// Copyright (c) 2024 Loupe (https://loupe.team), provided under the MIT License.

INTERFACE IPLCopenCommand

METHOD Aborted : BOOL
VAR_INPUT
END_VAR
END_METHOD

METHOD AbortPreviousCommands : BOOL
VAR_INPUT
    newCommand : IPLCopenCommand;
END_VAR
END_METHOD

PROPERTY Consume : BOOL
GET
END_GET
END_PROPERTY

METHOD Errored : BOOL
VAR_INPUT
    ID : INT;
END_VAR
END_METHOD

PROPERTY Execute : BOOL
SET
END_SET
END_PROPERTY

METHOD Finished : BOOL
VAR_INPUT
END_VAR
END_METHOD

METHOD RegisterGroup : BOOL
VAR_INPUT
    group : IPLCopenGroup;
END_VAR
END_METHOD

{warning 'add property implementation'}
PROPERTY Remote : IPLCopenCall
GET
END_GET
SET
END_SET
END_PROPERTY

PROPERTY Status : PLCopenStatusBase
GET
END_GET
END_PROPERTY

END_INTERFACE

(* stored: Version 1.1.0.1
   Itf IPLCopenCommand: Id {b8a2e96e-644a-4a58-85de-dacd7b91c166}
   Method Aborted: Id {9d6d52ef-ef78-446b-8945-f54bce7d4c7d}
   Method AbortPreviousCommands: Id {118dd5ed-57aa-4c07-ad44-4088eeac9e5c}
   Property Consume: Id {964841b7-219f-4d91-abbc-4e694a63fbfd}
   Get Get: Id {4e535252-1866-4d3a-84c2-c265027de691}
   Method Errored: Id {555f5ff6-f7de-4a4d-96f0-5c1829a76433}
   Property Execute: Id {191d42b1-9768-413a-8dd5-5e2df0572dc2}
   Set Set: Id {c1c106ad-262f-465b-9bb4-b6e1e214a2e2}
   Method Finished: Id {8d4ad453-b5db-4cb5-9fad-fde134f92b71}
   Method RegisterGroup: Id {75eeace0-1636-4dbc-8de2-8401cd2ef881}
   Property Remote: Id {57e041e0-47dd-412b-8e3f-60bcf4f3351e}
   Get Get: Id {d280f6d0-bd45-4d6a-bf59-884213c7b933}
   Set Set: Id {111b980b-e4e5-4722-9a7e-2393b1af29cb}
   Property Status: Id {19a8f19b-6eef-4123-af85-596f1682d840}
   Get Get: Id {4d51c448-5bf2-40e3-9b67-57a69f90d56b} *)
